Omron CX-Programmer project NewProject (CX-Programmer 9.81)

# PLC NewPLC1: CJ2M CPU11

## Program NewProgram1 (cyclic task 0)
Local symbols
BE 0.00 BOOL  ; Botão Emergência
BS 0.01 BOOL  ; Botão Stop
BST 0.02 BOOL  ; Botão Start
KM1 1.00 BOOL  ; Contactor 1
KM2 1.01 BOOL  ; Contactor 2
NO2KM1 1.00 BOOL  ; Segundo NO do KM1
NOKM1 1.00 BOOL  ; NO do Km1
NOKM2 1.01 BOOL  ; NO do Km2

### Section Section1

### Section OUTPUTS

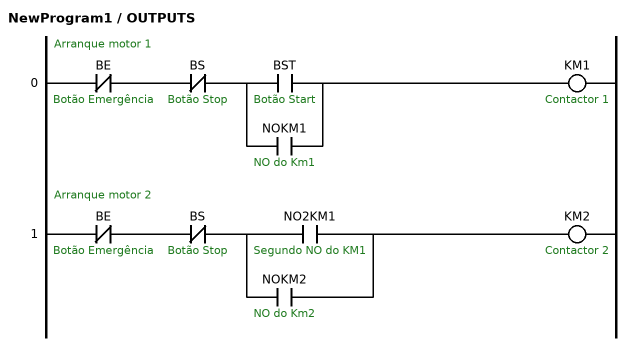
; rung 0: Arranque motor 1
LDNOT BE  ; Botão Emergência
ANDNOT BS  ; Botão Stop
LD BST  ; Botão Start
OR NOKM1  ; NO do Km1
ANDLD
OUT KM1  ; Contactor 1
; rung 1: Arranque motor 2
LDNOT BE  ; Botão Emergência
ANDNOT BS  ; Botão Stop
LD NO2KM1  ; Segundo NO do KM1
OR NOKM2  ; NO do Km2
ANDLD
OUT KM2  ; Contactor 2

### Section END
; rung 0
END(001)